{attribute 'obsolete' := 'Use E_StageEnableMode'}
TYPE ENUM_StageEnableMode : E_StageEnableMode; END_TYPE

(* stored: Version 1.1.0.1
   DUT ENUM_StageEnableMode: Id {43aedf2d-0b75-40d5-bd71-67b45334628a} *)
